TYPE CyclicAxis_CMD_typ :
STRUCT
		
	CyclicPos : CyclicPos_CMD_typ;
	CyclicVel : CyclicVel_CMD_typ;		
	
END_STRUCT
END_TYPE

(* stored: Version 1.1.0.1, ProductVersion 3.1.4024.3
   DUT CyclicAxis_CMD_typ: Id {b0157640-8a3e-0d4b-1ff9-90e320140116} *)
